FUNCTION_BLOCK NC_Axis EXTENDS TE_AxisBase0
VAR_INPUT
	enable		: BOOL;
	reset		: BOOL;
	home		: BOOL;
	refPos		: LREAL;
END_VAR
VAR_OUTPUT
	ready		: BOOL;
	enabled		: BOOL;
	referenced	: BOOL;
	error		: BOOL;
END_VAR
VAR
	ncRef		: AXIS_REF;
	ncPower		: MC_Power;
	ncReset		: MC_Reset;
	drvHoming	: DriveControlledHoming;
END_VAR


ncPower.Enable			:= enable;
ncPower.Enable_Negative	:= TRUE;
ncPower.Enable_Positive	:= TRUE;
ncPower(Axis:= ncRef);

ncReset.Execute := reset;
ncReset(Axis := ncRef);

ncRef.ReadStatus();

enabled := ncRef.Status.ControlLoopClosed AND ncRef.Status.Operational;
referenced := ncRef.Status.Homed;
error := ncRef.Status.Error;

(* drive controlled homing *)
drvHoming.execute := home;
drvHoming.refPos := refPos;
drvHoming(axis := THIS^, axisRef := ncRef);

(* This handles errors (error=TRUE) and warnings (error=FALSE) as TwinCat message *)
CallSlow();

END_FUNCTION_BLOCK

(* stored: Version 1.1.0.1, ProductVersion 3.1.4024.12
   POU NC_Axis: Id {281dffcb-fc8d-4de7-92f3-a0cb595f572d}, SpecialFunc None *)
